FUNCTION_BLOCK FB_DeclineNcConveyer IMPLEMENTS  I_NcConveyer
VAR_INPUT
END_VAR
VAR_OUTPUT
END_VAR
VAR
	_Axis1	: AXIS_REF;
	_Axis2	: AXIS_REF;
	
END_VAR

{warning 'add property implementation'}
PROPERTY Axis1 : Tc2_MC2.AXIS_REF
GET
Axis1 := _Axis1;
END_GET
SET
_Axis1 := Axis1;
END_SET
END_PROPERTY

{warning 'add property implementation'}
PROPERTY Axis2 : Tc2_MC2.AXIS_REF
GET
Axis2 := _Axis2;
END_GET
SET
_Axis2 := Axis2;
END_SET
END_PROPERTY

{warning 'add method implementation '}
METHOD Execute : BOOL
ADSLOGSTR(ADSLOG_MSGTYPE_LOG,'Moving Decline-Belt','');
END_METHOD

{warning 'add method implementation '}
METHOD Reset : BOOL
ADSLOGSTR(ADSLOG_MSGTYPE_LOG,'Reseting Decline','');
END_METHOD

{warning 'add method implementation '}
METHOD Start : BOOL
ADSLOGSTR(ADSLOG_MSGTYPE_LOG,'Powering Decline-Belt On','');
END_METHOD

{warning 'add method implementation '}
METHOD Stop : BOOL
ADSLOGSTR(ADSLOG_MSGTYPE_LOG,'Stopping Decline-Belt','');
END_METHOD

END_FUNCTION_BLOCK

(* stored: Version 1.1.0.1, ProductVersion 3.1.4024.6
   POU FB_DeclineNcConveyer: Id {c3a7c5d2-aac3-4959-952c-c4c0cf2187e3}, SpecialFunc None
   Property Axis1: Id {db2222ac-34a5-424a-a376-7652cf859b52}
   Get Get: Id {55fe05e3-1fe2-403e-bead-f69943d6d725}
   Set Set: Id {ef2ce5db-4da3-4bae-b6ee-fe9392eb1f00}
   Property Axis2: Id {813b03a9-dfa2-4f7a-8fd8-e77a3192c9f0}
   Get Get: Id {ce7fff66-4a2d-4a3c-a674-bc94c625de79}
   Set Set: Id {95481bc5-ce80-4bac-b67f-40749ec6b927}
   Method Execute: Id {313d9d47-1439-4ee9-9970-86bb2238d1a4}
   Method Reset: Id {7f51fbc5-debc-4758-a867-9387b4b0925c}
   Method Start: Id {d45d1a0e-5084-4fc6-951f-6b4983057d8b}
   Method Stop: Id {f16b825c-db0d-41aa-aae8-64a00f870648} *)
